(* PLC project PID, Beckhoff Automation GmbH TwinCAT PLC Control 3.5.13.21 *)
(* stored: creationDateTime 2022-05-17T15:59:31.94722, modificationDateTime 2022-05-17T15:59:31.94722 *)

{attribute 'qualified_only'}
{attribute 'strict'}
TYPE E_System_Mode :
(
	System_Init := 0,
	System_Run
);
END_TYPE
